FUNCTION CheckCalculation : LREAL
VAR_INPUT
  otg : REFERENCE TO Struckig.Ruckig;
END_VAR

REPEAT 
  otg();
  otg.CurrentPosition := otg.NewPosition;
  otg.CurrentVelocity := otg.NewVelocity;
  otg.CurrentAcceleration := otg.NewAcceleration;
UNTIL otg.State <> Struckig.TrajectoryState.busy END_REPEAT

CheckCalculation := otg.Duration;

END_FUNCTION

(* stored: Version 1.1.0.1, ProductVersion 3.1.4024.9
   POU CheckCalculation: Id {7705c60f-b3f4-4b53-bef5-2ced749a7c74}, SpecialFunc None *)
